(* CODESYS project PARTIDA_COM_TEMPO.project

Project tree, tasks and I/O mapping:
  Device : CODESYS Control Win V3, 3S - Smart Software Solutions GmbH, order no. 305021, version 3.5.11.30
    application Application
      libraries: Standard, * (System)
      task MainTask (cyclic, interval t#20ms, priority 1) calls PLC_PRG
      task VISU_TASK (cyclic, interval 100 ms, priority 31) calls VisuElems.Visu_Prg
      program PLC_PRG [LD]
      visualisation Visualization
  text list GlobalTextList
*)

// Device/Application/PLC_PRG
PROGRAM PLC_PRG
VAR
	START: BOOL;
	STOP: BOOL;
	TON_1: TON;
	MOTOR_1: BOOL;
	T0: TIME;
	TON_2: TON;
	T1: TIME;
	MOTOR_2: BOOL;
	MOTOR_3: BOOL;
	TON_3: TON;
	T3: TIME;
END_VAR

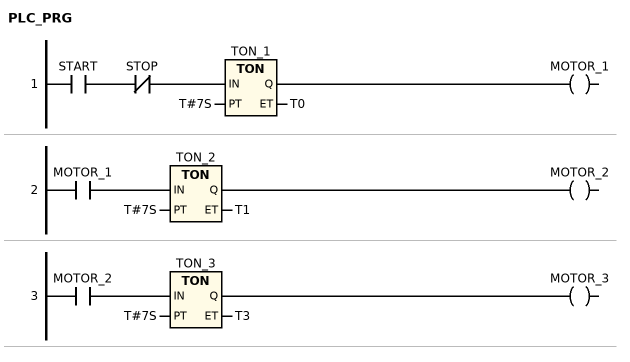
// NETWORK 1
TON_1(IN := START AND NOT STOP, PT := T#7S, ET => T0); // TON
MOTOR_1 := TON_1.Q;

// NETWORK 2
TON_2(IN := MOTOR_1, PT := T#7S, ET => T1); // TON
MOTOR_2 := TON_2.Q;

// NETWORK 3
TON_3(IN := MOTOR_2, PT := T#7S, ET => T3); // TON
MOTOR_3 := TON_3.Q;

END_PROGRAM

// Device/Application/Visualization
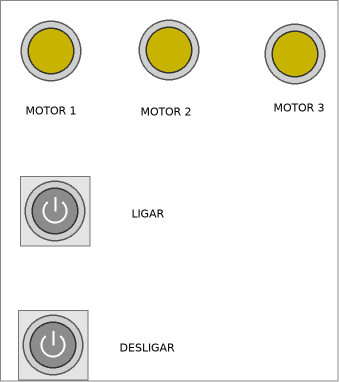
VISUALIZATION Visualization  // 339x382
    Lamp1 (16,16 70x70), variable: PLC_PRG.MOTOR_1, style: Lamp-Lamp1-Yellow
    Lamp1 (260,19 70x70), variable: PLC_PRG.MOTOR_3, style: Lamp-Lamp1-Yellow
    Lamp1 (134,15 70x70), variable: PLC_PRG.MOTOR_2, style: Lamp-Lamp1-Yellow
    PowerSwitch (20,176 70x70), variable: PLC_PRG.START, behaviour: TOGGLE, style: Switch-PowerSwitch-Gray
    PowerSwitch (18,310 70x70), variable: PLC_PRG.STOP, behaviour: TOGGLE, style: Switch-PowerSwitch-Gray
    Label (13,96 76x30), "MOTOR 1"
    Label (128,97 76x30), "MOTOR 2"
    Label (261,93 76x30), "MOTOR 3"
    Label (110,199 76x30), "LIGAR"
    Label (109,333 76x30), "DESLIGAR"
END_VISUALIZATION
